{attribute 'GeneratedUsingTerminal: EL6631-0000-0016'}
{attribute addProperty BoxType "EL6631-0000-0016"}
{attribute addProperty Id "EtcSlaveTerminalBaseInfoDataAT %I*InfoData_90184F0C16"}
{attribute addProperty CRC "354618671"}
{attribute addProperty Size "16"}
TYPE EL6631_15230D2F EXTENDS EtcSlaveTerminalBase :
STRUCT
	{attribute addProperty Name "InfoData"}
	InfoData : InfoData_90184F0C;
END_STRUCT
END_TYPE

(* stored: Version 1.2.0.0, ProductVersion 3.1.4024.9
   DUT EL6631_15230D2F: Id {4d8eb40c-4cbb-483d-a1a0-fc0d48ab5512} *)
